// TIA Portal V19 export
DATA_BLOCK "System_IDB"   // DB11
{ DB_Accessible_From_OPC_UA := 'FALSE' }
AUTHOR : Piemme
FAMILY : System
VERSION : 1.2
// stored: DBAccessibleFromOPCUA false, InstanceOfName System_FB, InstanceOfType FB
"System_FB"
   // VAR_INPUT
   //    PbLampTest : Bool;
   // END_VAR
   // VAR
   //    Ton0 : IEC_TIMER;
   //    wFrequencyGen : Word;
   //    wFrequencyLampTest : Word;
   //    PreviuosCycleTime : "CpuPreviuosCycleTime";
   // END_VAR
BEGIN
END_DATA_BLOCK
